{attribute 'TcGenerated'}
{attribute 'no-analysis'}
{attribute 'linkalways'}
// This function has been automatically generated from the project information.
VAR_GLOBAL CONSTANT
	{attribute 'const_non_replaced'}
	stLibVersion_FsControllerToolbox : ST_LibVersion := (iMajor := 0, iMinor := 4, iBuild := 0, iRevision := 0, nFlags := 0, sVersion := '0.4.0');
END_VAR

(* stored: Version 1.1.0.1, ProductVersion 3.1.4024.15
   GVL Global_Version: Id {73d8c8d8-6907-46c8-9d59-1d8f8d8defd2} *)
